PROGRAM MAIN
VAR
END_VAR

END_PROGRAM

(* stored: Version 1.1.0.1
   POU MAIN: Id {0c255287-5c04-4318-ae35-4538afeb31e9} *)
